Staubli VAL3: onExit.pgx

program onExit(bool x_bSave)
begin
// on exit
  if x_bSave
    axis:libSave()
  endIf
end
